FUNCTION_BLOCK F_OR (* standard bitwise boolean OR function *)
  (* Standard: 61131-3; Classification: standard bitwise boolean function; Description: Copyright (c) 2011 TU Wien ACIN This program and the accompanying materials are made available under the terms of the Eclipse Public License 2.0 which is available at https://www.eclipse.org/legal/epl-2.0/ SPDX-License-Identifier: EPL-2.0 *)
  (* Version 1.0, 2011-06-21, Monika Wenger, TU Wien ACIN *)
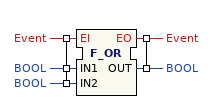
  EVENT_INPUT
    EI WITH IN1, IN2; (* Service Request *)
  END_EVENT
  EVENT_OUTPUT
    EO WITH OUT; (* Confirmation of Requested Service *)
  END_EVENT
  VAR_INPUT
    IN1 : BOOL; (* Input *)
    IN2 : BOOL; (* Input *)
  END_VAR
  VAR_OUTPUT
    OUT : BOOL; (* Output *)
  END_VAR
END_FUNCTION_BLOCK
